{attribute 'GeneratedUsingTerminal: EL5151-0080-0016'}
{attribute addProperty BoxType "EL5151-0080-0016"}
{attribute addProperty Id "EtcSlaveTerminalBaseENC_InputsAT %I*ENC_Inputs_F139456B14ENC_Inputs_1AT %I*ENC_Inputs_24B63C534ENC_OutputsAT %Q*ENC_Outputs_6FDDC6696WcStateAT %I*WcState_9091E0EB2InfoDataAT %I*InfoData_32EB74EA10"}
{attribute addProperty CRC "4224683339"}
{attribute addProperty Size "36"}
TYPE EL5151_FBCF8D4B EXTENDS EtcSlaveTerminalBase :
STRUCT
	{attribute addProperty Name "ENC_Inputs"}
	ENC_Inputs : ENC_Inputs_F139456B;
	{attribute addProperty Name "ENC_Inputs_1"}
	ENC_Inputs_1 : ENC_Inputs_24B63C53;
	{attribute addProperty Name "ENC_Outputs"}
	ENC_Outputs : ENC_Outputs_6FDDC669;
	{attribute addProperty Name "WcState"}
	WcState : WcState_9091E0EB;
	{attribute addProperty Name "InfoData"}
	InfoData : InfoData_32EB74EA;
END_STRUCT
END_TYPE

(* stored: Version 1.2.0.0, ProductVersion 3.1.4024.9
   DUT EL5151_FBCF8D4B: Id {b535f98b-7367-4915-8837-0e82725b60c1} *)
